Fanuc KAREL source: kt00442.KL

-- PROVISIONAL review KL for V1013-1; original PC SHA256 b4b1620966ef387f8c969ee5a001296b5e0e7b1226282942ee1fca533362fddb
-- Incomplete behavior may be omitted. Consult companion uncertainty JSON. Do not deploy.
PROGRAM KT00442
%NOLOCKGROUP
VAR
  R1 : REAL
  R2 : REAL
  OUT : BOOLEAN
BEGIN
  -- UNRESOLVED_PC offsets 5-16; opcodes 2E,23
  -- UNRESOLVED_PC offsets 21-32; opcodes 2E,23
  -- UNRESOLVED_PC offsets 37-48; opcodes 2E,23
  -- UNRESOLVED_PC offsets 53-64; opcodes 2E,23
  -- UNRESOLVED_PC offsets 69-88; opcodes 21,21,72,23
  -- UNRESOLVED_PC offsets 93-97; opcodes 7F
END KT00442
